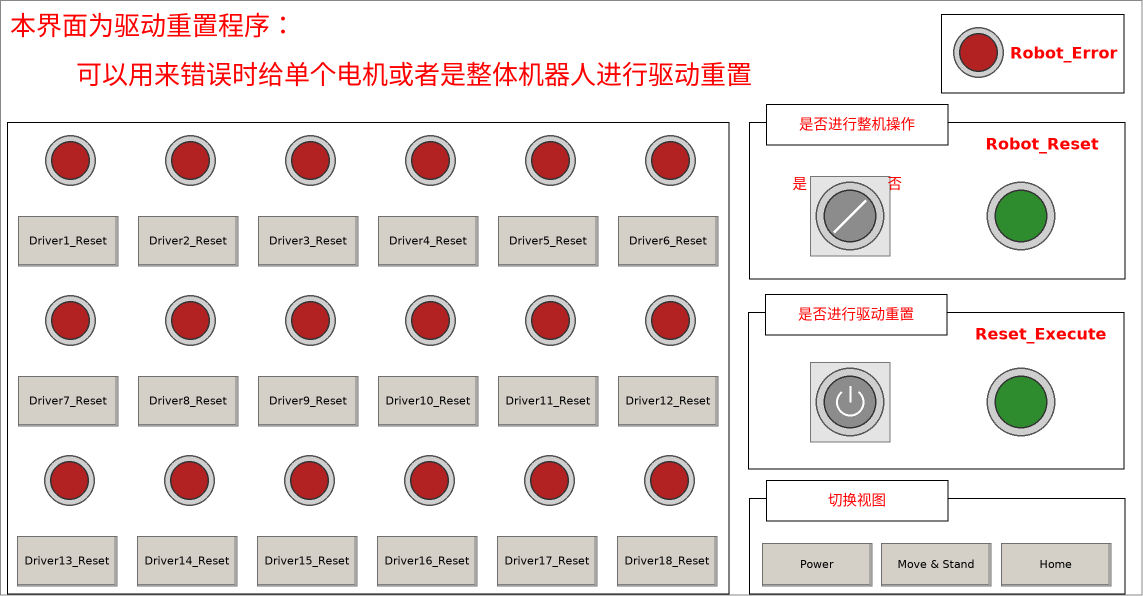
VISUALIZATION Visu_Reset  // 1143x596
    Rectangle (7,122 722x472)
    Lamp1 (40,131 61x59), variable: MAIN.Axis_Error[1], style: Lamp-Lamp1-Red
    Lamp1 (160,131 61x59), variable: MAIN.Axis_Error[2], style: Lamp-Lamp1-Red
    Lamp1 (280,131 61x59), variable: MAIN.Axis_Error[3], style: Lamp-Lamp1-Red
    Lamp1 (400,131 61x59), variable: MAIN.Axis_Error[4], style: Lamp-Lamp1-Red
    Lamp1 (520,131 61x59), variable: MAIN.Axis_Error[5], style: Lamp-Lamp1-Red
    Lamp1 (640,131 61x59), variable: MAIN.Axis_Error[6], style: Lamp-Lamp1-Red
    Button (18,216 100x50), "Driver1_Reset"
        tap MAIN.Axis_Reset[1]
    Button (138,216 100x50), "Driver2_Reset"
        tap MAIN.Axis_Reset[2]
    Button (258,216 100x50), "Driver3_Reset"
        tap MAIN.Axis_Reset[3]
    Button (378,216 100x50), "Driver4_Reset"
        tap MAIN.Axis_Reset[4]
    Button (498,216 100x50), "Driver5_Reset"
        tap MAIN.Axis_Reset[5]
    Button (618,216 100x50), "Driver6_Reset"
        tap MAIN.Axis_Reset[6]
    Lamp1 (40,291 61x59), variable: MAIN.Axis_Error[7], style: Lamp-Lamp1-Red
    Lamp1 (160,291 61x59), variable: MAIN.Axis_Error[8], style: Lamp-Lamp1-Red
    Lamp1 (280,291 61x59), variable: MAIN.Axis_Error[9], style: Lamp-Lamp1-Red
    Lamp1 (400,291 61x59), variable: MAIN.Axis_Error[10], style: Lamp-Lamp1-Red
    Lamp1 (520,291 61x59), variable: MAIN.Axis_Error[11], style: Lamp-Lamp1-Red
    Lamp1 (640,291 61x59), variable: MAIN.Axis_Error[12], style: Lamp-Lamp1-Red
    Button (18,376 100x50), "Driver7_Reset"
        tap MAIN.Axis_Reset[7]
    Button (138,376 100x50), "Driver8_Reset"
        tap MAIN.Axis_Reset[8]
    Button (258,376 100x50), "Driver9_Reset"
        tap MAIN.Axis_Reset[9]
    Button (378,376 100x50), "Driver10_Reset"
        tap MAIN.Axis_Reset[10]
    Button (498,376 100x50), "Driver11_Reset"
        tap MAIN.Axis_Reset[11]
    Button (618,376 100x50), "Driver12_Reset"
        tap MAIN.Axis_Reset[12]
    Lamp1 (39,451 61x59), variable: MAIN.Axis_Error[13], style: Lamp-Lamp1-Red
    Lamp1 (159,451 61x59), variable: MAIN.Axis_Error[14], style: Lamp-Lamp1-Red
    Lamp1 (279,451 61x59), variable: MAIN.Axis_Error[15], style: Lamp-Lamp1-Red
    Lamp1 (399,451 61x59), variable: MAIN.Axis_Error[16], style: Lamp-Lamp1-Red
    Lamp1 (519,451 61x59), variable: MAIN.Axis_Error[17], style: Lamp-Lamp1-Red
    Lamp1 (639,451 61x59), variable: MAIN.Axis_Error[18], style: Lamp-Lamp1-Red
    Button (17,536 100x50), "Driver13_Reset"
        tap MAIN.Axis_Reset[13]
    Button (137,536 100x50), "Driver14_Reset"
        tap MAIN.Axis_Reset[14]
    Button (257,536 100x50), "Driver15_Reset"
        tap MAIN.Axis_Reset[15]
    Button (377,536 100x50), "Driver16_Reset"
        tap MAIN.Axis_Reset[16]
    Button (497,536 100x50), "Driver17_Reset"
        tap MAIN.Axis_Reset[17]
    Button (617,536 100x50), "Driver18_Reset"
        tap MAIN.Axis_Reset[18]
    Rectangle (749,122 376x157)
    Label (965,128 154x32), "Robot_Reset"
    Rectangle (766,104 182x41), "是否进行整机操作"
    Rectangle (748,312 376x157)
    Label (964,318 154x32), "Reset_Execute"
    Rectangle (765,294 182x41), "是否进行驱动重置"
    Lamp1 (981,176 80x80), variable: MAIN.Robot_Reset, style: Lamp-Lamp1-Green
    Lamp1 (981,362 80x80), variable: MAIN.Reset_Execute, style: Lamp-Lamp1-Green
    RotarySwitch (810,176 80x80), variable: MAIN.Robot_Reset, behaviour: TOGGLE, style: Switch-RotarySwitch-Gray
    Rectangle (749,498 376x96)
    Rectangle (766,480 182x41), "切换视图"
    Label (865,169 60x30), "否"
    Label (770,169 60x30), "是"
    PowerSwitch (810,362 80x80), variable: MAIN.Reset_Execute, behaviour: TOGGLE, style: Switch-PowerSwitch-Gray
    Label (7,5 365x42), "本界面为驱动重置程序："
    Label (73,54 874x42), "可以用来错误时给单个电机或者是整体机器人进行驱动重置"
    Rectangle (941,14 183x79)
    Lamp1 (948,23 61x59), variable: MAIN.Robot_Error, style: Lamp-Lamp1-Red
    Label (987,37 154x32), "Robot_Error"
    Button (762,543 110x43), "Power"
        OnMouseClick: change screen: Visu_Power
    Button (1001,543 110x43), "Home"
        OnMouseClick: change screen: Visu_Home
    Button (881,543 110x43), "Move & Stand"
        OnMouseClick: change screen: Visu_Stand
END_VISUALIZATION

(* stored: Version 1.1.0.1, ProductVersion 3.1.4020.12
   Visu Visu_Reset: Id {a8fe9b11-4955-4a47-b72b-fe91df4e3617} *)
